Xinje XCPPro project, PLC1: XC2-42 (software 3.3q)

PROGRAM Ladder

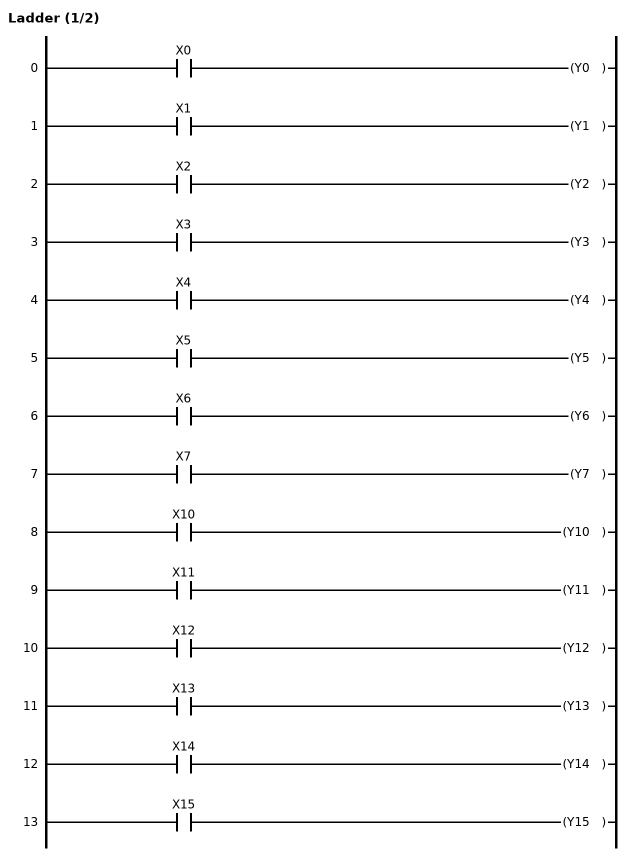
LD     X0
OUT    Y0
LD     X1
OUT    Y1
LD     X2
OUT    Y2
LD     X3
OUT    Y3
LD     X4
OUT    Y4
LD     X5
OUT    Y5
LD     X6
OUT    Y6
LD     X7
OUT    Y7
LD     X10
OUT    Y10
LD     X11
OUT    Y11
LD     X12
OUT    Y12
LD     X13
OUT    Y13
LD     X14
OUT    Y14
LD     X15
OUT    Y15

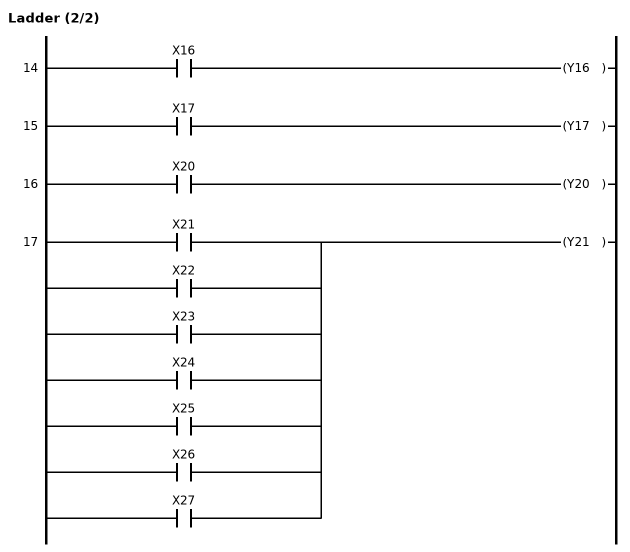
LD     X16
OUT    Y16
LD     X17
OUT    Y17
LD     X20
OUT    Y20
LD     X21
OR     X22
OR     X23
OR     X24
OR     X25
OR     X26
OR     X27
OUT    Y21